TEXTLIST TL_FbStateMUTING
  0 = 'UNDEFINED'
  1 = 'RUN'
  2 = 'STOP'
  3 = 'SAFE'
  4 = 'ERROR'
  5 = 'RESET'
  8 = 'DELAY OUT'
  9 = 'MUTING 1'
  10 = 'MUTING 2'
  11 = 'MUTING 3'
  12 = 'MUTING 4'
  13 = 'MUTING 5'
  14 = 'MUTING 6'
  15 = 'MUTING 7'
  16 = 'MUTING 8'
  17 = 'MUTING 9'
   = ''
END_TEXTLIST

(* stored: Version 1.1.0.1, ProductVersion 3.1.4022.12
   TextList TL_FbStateMUTING: Id {286014ae-0a21-4e52-bda6-44fbfa45ae7f} *)
